FUNCTION XNOR : BOOL
VAR_INPUT
	A	:	BOOL;
	B	:	BOOL;
END_VAR
VAR
END_VAR

XNOR := (A AND B) OR ((NOT A) AND  (NOT B));

END_FUNCTION

(* stored: Version 1.1.0.1, ProductVersion 3.1.4024.15
   POU XNOR: Id {effdb1b1-0512-4630-a66b-8b98029bf13e}, SpecialFunc None *)
